FUNCTION F_CutInstancePath : STRING(512)
VAR_INPUT
	sSrc			:STRING(512);
END_VAR
VAR
	sDelimiter		:STRING(1) := '.';
	iFnd			:UDINT;
	sSubstr			:STRING(512);
END_VAR

// sSrc := 'TE_SP_Module_Demo.TE_SP_Module_Demo_PlcRt1.P_MachineSet.fbMa2.fbDemoSequence.fbLenzei550';

iFnd := FIND2(ADR(sSrc), ADR(sDelimiter));
IF (iFnd > 0) THEN
	DELETE2(ADR(sSrc), ADR(sSubstr), SIZEOF(sSubstr), iFnd, 1);
END_IF
iFnd := FIND2(ADR(sSubstr), ADR(sDelimiter));
IF (iFnd > 0) THEN
	DELETE2(ADR(sSubstr), ADR(sSubstr), SIZEOF(sSubstr), iFnd, 1);
END_IF

F_CutInstancePath := sSubstr;

END_FUNCTION

(* stored: Version 1.1.0.1, ProductVersion 3.1.4024.11
   POU F_CutInstancePath: Id {063e07bb-5db6-4428-a76f-99ab182ae752}, SpecialFunc None *)
